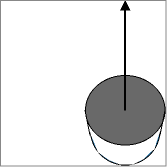
VISUALIZATION VISU_Tube_Top_2  // 167x167
VAR_IN_OUT
	azi : LREAL;
END_VAR
    Ellipse (90,95 70x70)
        p2858320360: azi
    Polygon (85,115) (165,115) (156,142) (154,149) (150,152) (143,159) (133,164) (119,164) (109,160) (98,152) (91,135)
        p2858320360: azi
    Ellipse (85,75 80x70)
        p2858320360: azi
    Polygon (120,10) (125,0) (130,10)
        p2858320360: azi
    Polyline (125,110) (125,10)
        p2858320360: azi
    Polyline (160,135) (165,110)
        p2858320360: azi
    Polyline (90,135) (85,110)
        p2858320360: azi
END_VISUALIZATION

(* stored: Version 1.1.0.1, ProductVersion 3.1.4018.5
   Visu VISU_Tube_Top_2: Id {6f826252-2719-4300-964c-14fbc636f840} *)
